FUNCTION_BLOCK XtsMoverAxis EXTENDS CyclicBase
VAR
	MyAxisRef : AXIS_REF;
	_MyAxisStatus : ST_AxisStatus;
	_MyNCData : NCTOPLC_AXIS_REF;
	MoverPowerCommand : AxisPower(MyAxisRef);
	MoverMoveCommand : MoveModuloMoverToPosition(MyAxisRef) := (Gap := 100.0);
	MoverHaltCommand : HaltMover(MyAxisRef);
	MoverResetCommand : AxesReset(MyAxisRef);
	MoverActivateTrackCommand : ActivateTrackForMover(MyAxisRef);
	_ipTcIoXtsMover	: I_TcIoXtsXpuMover;
	_ActiveTrackLength : MC_LREAL;
	TrackChangeTrigger : R_TRIG;
	//axesMoveModuloTo 		: MoveModuloMoverToPosition(_Axis) := (Gap := 100.0);
	_MoverAbsMoveOptions : ST_MoveAbsoluteCAOptions;
	_stTmsActPositions			: ST_PositionInfo;
END_VAR
VAR CONSTANT
	_MaxMoverVelocity : MC_LREAL := 4000.0;
END_VAR

PROPERTY PUBLIC Acceleration : MC_LREAL
GET
Acceleration := MoverMoveCommand.Acceleration;
END_GET
SET
MoverMoveCommand.Acceleration := Acceleration;
END_SET
END_PROPERTY

METHOD ActivateTrack : HRESULT
VAR_INPUT
	NewTrack : OTCID;
END_VAR
IF NOT MoverActivateTrackCommand.Busy AND THIS^.isMoverStationary() AND NewTrack <> 0  THEN
	IF MoverActivateTrackCommand.Execute(Track := NewTrack) THEN
		ResetAxis := 1;
	ELSE
		ResetAxis := -1;
	END_IF
ELSE
	ResetAxis := -1;
END_IF
END_METHOD

METHOD PUBLIC  Cycle : HRESULT
VAR_INPUT
END_VAR
IF isMoverDetected() THEN
	MyAxisRef.ReadStatus();
	_MyAxisStatus := MyAxisRef.Status;
	_MyNCData := MyAxisRef.NcToPlc;
	MoverPowerCommand.Cycle();
	MoverMoveCommand.Cycle();
	MoverHaltCommand.Cycle();
	MoverResetCommand.Cycle();
	MoverActivateTrackCommand.Cycle();
	TrackChangeTrigger(CLK := MoverActivateTrackCommand.Done);
	IF TrackChangeTrigger.Q THEN
		_MoverAbsMoveOptions.PositionReferenceSystem :=  MoverActivateTrackCommand.NewTrackId;
		MoverMoveCommand.Options := _MoverAbsMoveOptions;
	END_IF
	IF _ipTcIoXtsMover <> 0 THEN
		_stTmsActPositions := _ipTcIoXtsMover.GetPositionInfo();
	END_IF
	Cycle := 1;
ELSE
	Cycle := -1;
END_IF
END_METHOD

PROPERTY PUBLIC Deceleration : MC_LREAL
GET
Deceleration := MoverMoveCommand.Deceleration;
END_GET
SET
MoverMoveCommand.Deceleration := MoverHaltCommand.Deceleration := Deceleration;
END_SET
END_PROPERTY

METHOD PUBLIC DisableMover : HRESULT
VAR_INPUT
END_VAR
IF THIS^.isMoverEnabled() AND NOT MoverPowerCommand.Busy THEN
	MoverPowerCommand.Disable();
	DisableMover := 1;
ELSE
	DisableMover := -1;
END_IF
END_METHOD

METHOD PUBLIC EnableMover : HRESULT
VAR_INPUT
END_VAR
IF (NOT MoverPowerCommand.Busy) AND NOT THIS^.isMoverEnabled() THEN
	MoverPowerCommand.Enable();
	EnableMover := 1;
ELSE
	EnableMover := -1;
END_IF
END_METHOD

METHOD FB_init : BOOL
VAR_INPUT
	bInitRetains : BOOL; // if TRUE, the retain variables are initialized (warm start / cold start)
	bInCopyCode : BOOL;  // if TRUE, the instance afterwards gets moved into the copy code (online change)
	XtsRunner : I_ObjectRunner;
END_VAR
XtsRunner.AddComponent(THIS^);
END_METHOD

PROPERTY PUBLIC Gap : MC_LREAL
GET
Gap := MoverMoveCommand.Gap;
END_GET
SET
IF Gap >= 50.0 THEN
	MoverMoveCommand.Gap := MoverHaltCommand.Gap := Gap;
ELSE
	Gap := 100.0;
END_IF
END_SET
END_PROPERTY

METHOD PUBLIC HaltAxis : HRESULT
VAR_INPUT
END_VAR
IF NOT MoverHaltCommand.Busy AND NOT THIS^.isMoverStationary() THEN
	IF MoverHaltCommand.Execute() THEN
		HaltAxis := 1;
	ELSE
		HaltAxis := -1;
	END_IF
ELSE
	HaltAxis := -1;
END_IF
END_METHOD

PROPERTY PUBLIC IdentInGroup : IDENT_IN_GROUP_REF
GET
IdentInGroup := UDINT_TO_IDENTINGROUP(id := _MyNCData.AxisId);
END_GET
END_PROPERTY

METHOD PUBLIC isMoverAtPosition : BOOL
VAR_INPUT
END_VAR
END_METHOD

METHOD PUBLIC isMoverDetected : BOOL
VAR_INPUT
END_VAR
isMoverDetected := _MyNCData.AxisId <> 0;
END_METHOD

METHOD PUBLIC isMoverEnabled : BOOL
VAR_INPUT
END_VAR
isMoverEnabled :=  NOT _MyAxisStatus.Disabled;
END_METHOD

METHOD PUBLIC isMoverStationary : BOOL
VAR_INPUT
END_VAR
isMoverStationary := _MyAxisStatus.NotMoving;
END_METHOD

PROPERTY PUBLIC Jerk : MC_LREAL
GET
Jerk := MoverMoveCommand.Jerk;
END_GET
SET
MoverMoveCommand.Jerk := MoverHaltCommand.Jerk := Jerk;
END_SET
END_PROPERTY

PROPERTY PUBLIC MoverErrorID : DWORD
GET
MoverErrorID := _MyAxisStatus.ErrorID;
END_GET
END_PROPERTY

PROPERTY PUBLIC MoversActiveTrack : OTCID
GET
MoversActiveTrack := _ipTcIoXtsMover.GetActiveTrackObjectId();
END_GET
END_PROPERTY

PROPERTY PUBLIC MoverXtsIoEnvInterface : I_TcIoXtsXpuMover
GET
MoverXtsIoEnvInterface := _ipTcIoXtsMover;
END_GET
SET
_ipTcIoXtsMover := MoverXtsIoEnvInterface;
END_SET
END_PROPERTY

METHOD PUBLIC MoveTo : HRESULT
VAR_INPUT
	RequiredPosition : MC_LREAL;
	MoveVelocity : MC_LREAL;
END_VAR
IF NOT MoverMoveCommand.Busy AND MoveVelocity < _MaxMoverVelocity AND RequiredPosition < _ActiveTrackLength AND Gap >= 50.0 THEN
	IF THIS^.MoverMoveCommand.MoveTo(Position := RequiredPosition, 
									Velocity := MoveVelocity, 
									Direction := Tc3_Mc3Definitions.MC_DIRECTION.mcDirectionPositive, 
									Turns := 0) THEN
									
		MoveTo := 1;
	END_IF
ELSE
	MoveTo := -1;
END_IF
END_METHOD

METHOD PUBLIC ResetAxis : HRESULT
VAR_INPUT
END_VAR
IF NOT MoverResetCommand.Busy AND _MyAxisStatus.Error THEN
	IF MoverResetCommand.Execute() THEN
		ResetAxis := 1;
	ELSE
		ResetAxis := -1;
	END_IF
ELSE
	ResetAxis := -1;
END_IF
END_METHOD

END_FUNCTION_BLOCK

(* stored: Version 1.1.0.1, ProductVersion 3.1.4024.12
   POU XtsMoverAxis: Id {f9a43ed2-0578-4aed-857c-1a3adef0c7f6}, SpecialFunc None
   Folder Administration: Id {660864df-8996-42d7-8e95-bfca1c90696e}
   Folder Commands: Id {db0a893b-cc1a-482e-a432-7e9d568c5112}
   Folder Dynamics: Id {6b49cc7a-c913-475a-9f9a-db91d65d07e1}
   Folder ICyclic: Id {895ad701-1670-4c6d-921e-cd7ccab0c12a}
   Folder Status: Id {b27ba391-8a3b-4e51-ae24-bae43a7b6e5f}
   Property Acceleration: Id {5cd04126-8ceb-4f9d-a4c5-c87e7e11d0e6}
   Get Get: Id {89c9e6d0-5dfa-4531-97de-32e16eb2e196}
   Set Set: Id {95cc2e62-d911-4757-83d0-b9b38a36fdde}
   Method ActivateTrack: Id {f7604675-5338-4e11-9132-b17d5df72cc8}
   Method Cycle: Id {b5956233-12ba-4cb8-805f-5693aec42bed}
   Property Deceleration: Id {3def2bbc-f7ec-4120-acb9-2ff2a2789bd5}
   Get Get: Id {e6097884-8279-4e20-92f9-6fb8b5120af4}
   Set Set: Id {dbf3cf03-c8db-40c9-ab3e-669bb5cdced1}
   Method DisableMover: Id {a82f95fa-77b4-4c5e-ae67-686dbd3b2d8d}
   Method EnableMover: Id {d130fe63-f34a-4455-8bb8-4dfcc482e573}
   Method FB_init: Id {b6181511-263e-44ed-9731-4c0d1e2c2029}
   Property Gap: Id {dd72da9d-fc94-421a-8ee7-a84a721dd20c}
   Get Get: Id {5c8fd02d-70e7-4f46-b386-6000a46a3487}
   Set Set: Id {280f9258-e1cd-43be-bf57-16929cbbc8d6}
   Method HaltAxis: Id {b177db81-8e99-498a-a7a2-cd0938dd7a2c}
   Property IdentInGroup: Id {4d5563a0-634a-4074-a0e4-612875dd790c}
   Get Get: Id {6419a53d-e416-464a-881c-e300db0a9add}
   Method isMoverAtPosition: Id {f1a74560-cd92-4fa6-83a2-3bacea608337}
   Method isMoverDetected: Id {c1a5811f-71c0-458a-bf03-7bfa946db86b}
   Method isMoverEnabled: Id {7f5530a3-9bf6-4669-8c7b-76814da68801}
   Method isMoverStationary: Id {64b09804-b6c0-46e5-9180-be650a88cf77}
   Property Jerk: Id {fbc5f504-aa6b-48f8-8a62-bbde3b74b20e}
   Get Get: Id {98c0c9db-aae6-4788-a223-2bf5fa007418}
   Set Set: Id {6a6a16a3-4f19-4f4d-bd8d-8441ae3b5cf2}
   Property MoverErrorID: Id {9a24b894-1b02-4293-95b1-831b38fd5fad}
   Get Get: Id {01f9b7c9-0e41-48f0-a5f9-8a7a495677b0}
   Property MoversActiveTrack: Id {15471ba0-8341-48c7-a2d0-01ca6286078a}
   Get Get: Id {2721855b-e1d8-4f74-a352-28794ee4ae69}
   Property MoverXtsIoEnvInterface: Id {6aaf98f4-e1bc-4f35-afbe-48664404e767}
   Get Get: Id {5b75808a-7c24-4c09-8809-4a555d5acdb1}
   Set Set: Id {57119448-dfbf-405e-ade1-72aad5224720}
   Method MoveTo: Id {ea6488b0-fefd-4f9f-a3b2-cfd8c6f64d05}
   Method ResetAxis: Id {e9d8249c-2f88-4980-a483-ceda82c7ab80} *)
